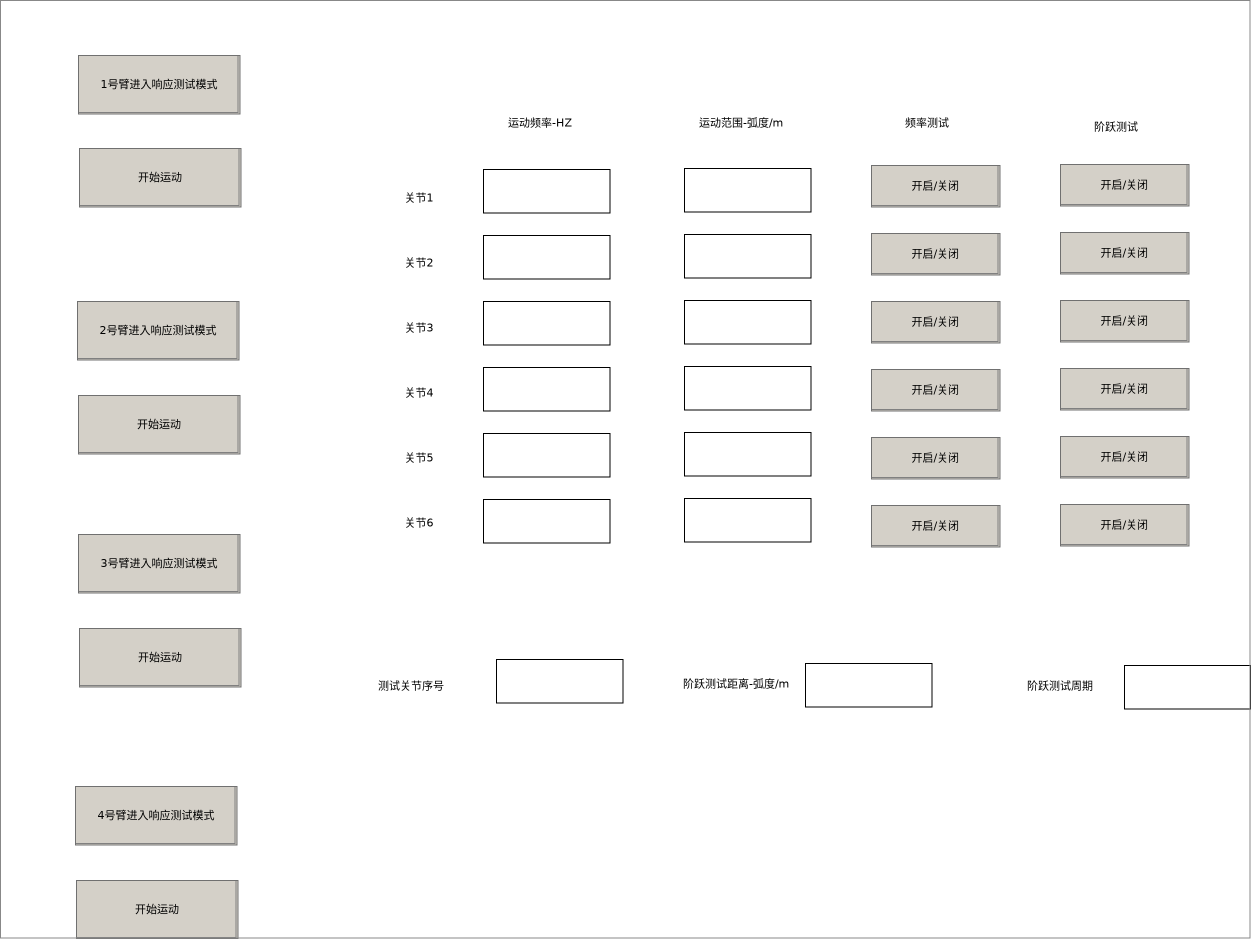
VISUALIZATION responseTest  // 1251x939
    Button (78,55 162x59), "1号臂进入响应测试模式", colour toggle: g_responseTest.m_testMode[1]
        toggle g_responseTest.m_testMode[1]
    Button (79,148 162x59), "开始运动", colour toggle: g_responseTest.m_startMotion[1]
        toggle g_responseTest.m_startMotion[1]
    Button (77,301 162x59), "2号臂进入响应测试模式", colour toggle: g_responseTest.m_testMode[2]
        toggle g_responseTest.m_testMode[2]
    Button (78,395 162x59), "开始运动", colour toggle: g_responseTest.m_startMotion[2]
        toggle g_responseTest.m_startMotion[2]
    Label (465,108 150x30), "运动频率-HZ"
    Label (666,108 150x30), "运动范围-弧度/m"
    Label (852,108 150x30), "频率测试"
    Label (1041,112 150x30), "阶跃测试"
    Label (344,183 150x30), "关节1"
    Label (344,248 150x30), "关节2"
    Label (344,313 150x30), "关节3"
    Label (344,378 150x30), "关节4"
    Label (344,443 150x30), "关节5"
    Label (344,508 150x30), "关节6"
    Rectangle (483,169 127x44), text variable: g_responseTest.m_jntMotionFreq[1]
        OnMouseClick: write the text variable via Default
    Rectangle (483,235 127x44), text variable: g_responseTest.m_jntMotionFreq[2]
        OnMouseClick: write the text variable via Default
    Rectangle (483,301 127x44), text variable: g_responseTest.m_jntMotionFreq[3]
        OnMouseClick: write the text variable via Default
    Rectangle (483,367 127x44), text variable: g_responseTest.m_jntMotionFreq[4]
        OnMouseClick: write the text variable via Default
    Rectangle (483,433 127x44), text variable: g_responseTest.m_jntMotionFreq[5]
        OnMouseClick: write the text variable via Default
    Rectangle (483,499 127x44), text variable: g_responseTest.m_jntMotionFreq[6]
        OnMouseClick: write the text variable via Default
    Rectangle (684,168 127x44), text variable: g_responseTest.m_jntMotionRange[1]
        OnMouseClick: write the text variable via Default
    Rectangle (684,234 127x44), text variable: g_responseTest.m_jntMotionRange[2]
        OnMouseClick: write the text variable via Default
    Rectangle (684,300 127x44), text variable: g_responseTest.m_jntMotionRange[3]
        OnMouseClick: write the text variable via Default
    Rectangle (684,366 127x44), text variable: g_responseTest.m_jntMotionRange[4]
        OnMouseClick: write the text variable via Default
    Rectangle (684,432 127x44), text variable: g_responseTest.m_jntMotionRange[5]
        OnMouseClick: write the text variable via Default
    Rectangle (684,498 127x44), text variable: g_responseTest.m_jntMotionRange[6]
        OnMouseClick: write the text variable via Default
    Button (871,165 129x42), "开启/关闭", colour toggle: g_responseTest.m_freqTestFlag[1]
        toggle g_responseTest.m_freqTestFlag[1]
    Button (871,233 129x42), "开启/关闭", colour toggle: g_responseTest.m_freqTestFlag[2]
        toggle g_responseTest.m_freqTestFlag[2]
    Button (871,301 129x42), "开启/关闭", colour toggle: g_responseTest.m_freqTestFlag[3]
        toggle g_responseTest.m_freqTestFlag[3]
    Button (871,369 129x42), "开启/关闭", colour toggle: g_responseTest.m_freqTestFlag[4]
        toggle g_responseTest.m_freqTestFlag[4]
    Button (871,437 129x42), "开启/关闭", colour toggle: g_responseTest.m_freqTestFlag[5]
        toggle g_responseTest.m_freqTestFlag[5]
    Button (871,505 129x42), "开启/关闭", colour toggle: g_responseTest.m_freqTestFlag[6]
        toggle g_responseTest.m_freqTestFlag[6]
    Button (1060,164 129x42), "开启/关闭", colour toggle: g_responseTest.m_stepTestFlag[1]
        toggle g_responseTest.m_stepTestFlag[1]
    Button (1060,232 129x42), "开启/关闭", colour toggle: g_responseTest.m_stepTestFlag[2]
        toggle g_responseTest.m_stepTestFlag[2]
    Button (1060,300 129x42), "开启/关闭", colour toggle: g_responseTest.m_stepTestFlag[3]
        toggle g_responseTest.m_stepTestFlag[3]
    Button (1060,368 129x42), "开启/关闭", colour toggle: g_responseTest.m_stepTestFlag[4]
        toggle g_responseTest.m_stepTestFlag[4]
    Button (1060,436 129x42), "开启/关闭", colour toggle: g_responseTest.m_stepTestFlag[5]
        toggle g_responseTest.m_stepTestFlag[5]
    Button (1060,504 129x42), "开启/关闭", colour toggle: g_responseTest.m_stepTestFlag[6]
        toggle g_responseTest.m_stepTestFlag[6]
    Label (336,671 150x30), "测试关节序号"
    Rectangle (496,659 127x44), text variable: g_responseTest.m_testJntIdx
        OnMouseClick: write the text variable via Default
    Label (661,669 150x30), "阶跃测试距离-弧度/m"
    Rectangle (805,663 127x44), text variable: g_responseTest.m_jntStep
        OnMouseClick: write the text variable via Default
    Label (985,671 150x30), "阶跃测试周期"
    Rectangle (1124,665 127x44), text variable: g_responseTest.m_stepCycle
        OnMouseClick: write the text variable via Default
    Button (78,534 162x59), "3号臂进入响应测试模式", colour toggle: g_responseTest.m_testMode[3]
        toggle g_responseTest.m_testMode[3]
    Button (79,628 162x59), "开始运动", colour toggle: g_responseTest.m_startMotion[3]
        toggle g_responseTest.m_startMotion[3]
    Button (75,786 162x59), "4号臂进入响应测试模式", colour toggle: g_responseTest.m_testMode[4]
        toggle g_responseTest.m_testMode[4]
    Button (76,880 162x59), "开始运动", colour toggle: g_responseTest.m_startMotion[4]
        toggle g_responseTest.m_startMotion[4]
END_VISUALIZATION

(* stored: Version 1.1.0.1, ProductVersion 3.1.4024.11
   Visu responseTest: Id {a42db8e4-fc1a-44c1-8e11-028315a58691} *)
